// TIA Portal V18 export
// export: Created 2026-01-09T11:31:58.8051596Z, ExportSetting WithDefaults, DisplayName Totally Integrated Automation Portal, DisplayVersion V18 Update 5, DisplayName TIA Portal Openness, DisplayVersion V18 Update 5, DisplayName TIA Portal Teamcenter Gateway, DisplayVersion V18, DisplayName TIA Portal Version Control Interface, DisplayVersion V18, DisplayName SINAMICS Startdrive Advanced, DisplayVersion V18 SP2 Update 1, DisplayName SINAMICS Startdrive G110M, G120, G120C, G120D, G120P, G115D, DisplayVersion V18 SP2 Update 1, DisplayName SINAMICS Startdrive G130, G150, S120, S150, SINAMICS MV, S210, G220, S200, DisplayVersion V18 SP2 Update 1, DisplayName STEP 7 Professional, DisplayVersion V18 Update 5, DisplayName STEP 7 Safety, DisplayVersion V18, DisplayName WinCC Professional, DisplayVersion V18 Update 5
TagTable "GlobalErrorWord"
  GlobalCOMError : Word  (%DB1066.DBW0, CPU S71500-2PN_TP700, 100 ms)
  PNSlaveStation01Error1 : Word  (%DB1066.DBW10, CPU S71500-2PN_TP700, 100 ms)
  PNSlaveStation01Error2 : Word  (%DB1066.DBW12, CPU S71500-2PN_TP700, 100 ms)
  PNSlaveStation01Error3 : Word  (%DB1066.DBW14, CPU S71500-2PN_TP700, 100 ms)
  PNSlaveStation01Error4 : Word  (%DB1066.DBW16, CPU S71500-2PN_TP700, 100 ms)
  PNSlaveStation01Error5 : Word  (%DB1066.DBW18, CPU S71500-2PN_TP700, 100 ms)
  PNSlaveStation01Error6 : Word  (%DB1066.DBW20, CPU S71500-2PN_TP700, 100 ms)
  PNSlaveStation01Error7 : Word  (%DB1066.DBW22, CPU S71500-2PN_TP700, 100 ms)
  PNSlaveStation01Error8 : Word  (%DB1066.DBW24, CPU S71500-2PN_TP700, 100 ms)
  PNSlaveStation01Error9 : Word  (%DB1066.DBW26, CPU S71500-2PN_TP700, 100 ms)
  PNSlaveStation01Error10 : Word  (%DB1066.DBW28, CPU S71500-2PN_TP700, 100 ms)
  SerialCOMM01Error : Word  (%DB1066.DBW30, CPU S71500-2PN_TP700, 100 ms)
  SerialCOMM02Error : Word  (%DB1066.DBW32, CPU S71500-2PN_TP700, 100 ms)
  SerialCOMM03Error : Word  (%DB1066.DBW34, CPU S71500-2PN_TP700, 100 ms)
  SerialCOMM04Error : Word  (%DB1066.DBW36, CPU S71500-2PN_TP700, 100 ms)
  SerialCOMM05Error : Word  (%DB1066.DBW38, CPU S71500-2PN_TP700, 100 ms)
  PNSlaveStation02Error1 : Word  (%DB1066.DBW40, CPU S71500-2PN_TP700, 100 ms)
  PNSlaveStation02Error2 : Word  (%DB1066.DBW42, CPU S71500-2PN_TP700, 100 ms)
  PNSlaveStation02Error3 : Word  (%DB1066.DBW44, CPU S71500-2PN_TP700, 100 ms)
  PNSlaveStation02Error4 : Word  (%DB1066.DBW46, CPU S71500-2PN_TP700, 100 ms)
  PNSlaveStation02Error5 : Word  (%DB1066.DBW48, CPU S71500-2PN_TP700, 100 ms)
  PNSlaveStation02Error6 : Word  (%DB1066.DBW50, CPU S71500-2PN_TP700, 100 ms)
  PNSlaveStation02Error7 : Word  (%DB1066.DBW52, CPU S71500-2PN_TP700, 100 ms)
  PNSlaveStation02Error8 : Word  (%DB1066.DBW54, CPU S71500-2PN_TP700, 100 ms)   // Fault: PLC_OP10_110A1_PNSlaveStationError
  PNSlaveStation02Error9 : Word  (%DB1066.DBW56, CPU S71500-2PN_TP700, 100 ms)
  PNSlaveStation02Error10 : Word  (%DB1066.DBW58, CPU S71500-2PN_TP700, 100 ms)
  PNSlaveStation03Error1 : Word  (%DB1066.DBW60, CPU S71500-2PN_TP700, 100 ms)
  PNSlaveStation03Error2 : Word  (%DB1066.DBW62, CPU S71500-2PN_TP700, 100 ms)
  PNSlaveStation03Error3 : Word  (%DB1066.DBW64, CPU S71500-2PN_TP700, 100 ms)
  PNSlaveStation03Error4 : Word  (%DB1066.DBW66, CPU S71500-2PN_TP700, 100 ms)
  PNSlaveStation03Error5 : Word  (%DB1066.DBW68, CPU S71500-2PN_TP700, 100 ms)
  PNSlaveStation03Error6 : Word  (%DB1066.DBW70, CPU S71500-2PN_TP700, 100 ms)
  PNSlaveStation03Error7 : Word  (%DB1066.DBW72, CPU S71500-2PN_TP700, 100 ms)
  PNSlaveStation03Error8 : Word  (%DB1066.DBW74, CPU S71500-2PN_TP700, 100 ms)
  PNSlaveStation03Error9 : Word  (%DB1066.DBW76, CPU S71500-2PN_TP700, 100 ms)
  PNSlaveStation03Error10 : Word  (%DB1066.DBW78, CPU S71500-2PN_TP700, 100 ms)
  ValveIsland01Error : Word  (%DB1066.DBW80, CPU S71500-2PN_TP700, 100 ms)
  ValveIsland02Error : Word  (%DB1066.DBW82, CPU S71500-2PN_TP700, 100 ms)
  ValveIsland03Error : Word  (%DB1066.DBW84, CPU S71500-2PN_TP700, 100 ms)
  ValveIsland04Error : Word  (%DB1066.DBW86, CPU S71500-2PN_TP700, 100 ms)
  ValveIsland05Error : Word  (%DB1066.DBW88, CPU S71500-2PN_TP700, 100 ms)
  SafetyGlobalError : Word  (%DB1066.DBW90, CPU S71500-2PN_TP700, 100 ms)
  SafetyDoorType01Error : Word  (%DB1066.DBW100, CPU S71500-2PN_TP700, 100 ms)
  SafetyDoorType02Error : Word  (%DB1066.DBW102, CPU S71500-2PN_TP700, 100 ms)
  SafetyDoorType03Error : Word  (%DB1066.DBW104, CPU S71500-2PN_TP700, 100 ms)
  SafetyDoorType04Error : Word  (%DB1066.DBW106, CPU S71500-2PN_TP700, 100 ms)
  SafetyDoorType05Error : Word  (%DB1066.DBW108, CPU S71500-2PN_TP700, 100 ms)
  SafetyDoor01Error : Word  (%DB1066.DBW110, CPU S71500-2PN_TP700, 100 ms)
  SafetyDoor02Error : Word  (%DB1066.DBW112, CPU S71500-2PN_TP700, 100 ms)
  SafetyDoor03Error : Word  (%DB1066.DBW114, CPU S71500-2PN_TP700, 100 ms)
  SafetyDoor04Error : Word  (%DB1066.DBW116, CPU S71500-2PN_TP700, 100 ms)
  SafetyDoor05Error : Word  (%DB1066.DBW118, CPU S71500-2PN_TP700, 100 ms)
  SafetyDoor06Error : Word  (%DB1066.DBW120, CPU S71500-2PN_TP700, 100 ms)
  SafetyDoor07Error : Word  (%DB1066.DBW122, CPU S71500-2PN_TP700, 100 ms)
  SafetyDoor08Error : Word  (%DB1066.DBW124, CPU S71500-2PN_TP700, 100 ms)
  SafetyDoor09Error : Word  (%DB1066.DBW126, CPU S71500-2PN_TP700, 100 ms)
  SafetyDoor10Error : Word  (%DB1066.DBW128, CPU S71500-2PN_TP700, 100 ms)
  LightCurtain01Error : Word  (%DB1066.DBW130, CPU S71500-2PN_TP700, 100 ms)
  LightCurtain02Error : Word  (%DB1066.DBW132, CPU S71500-2PN_TP700, 100 ms)
  LightCurtain03Error : Word  (%DB1066.DBW134, CPU S71500-2PN_TP700, 100 ms)
  LightCurtain04Error : Word  (%DB1066.DBW136, CPU S71500-2PN_TP700, 100 ms)
  LightCurtain05Error : Word  (%DB1066.DBW138, CPU S71500-2PN_TP700, 100 ms)
  Product01Error : Word  (%DB1066.DBW140, CPU S71500-2PN_TP700, 100 ms)
  Product02Error : Word  (%DB1066.DBW142, CPU S71500-2PN_TP700, 100 ms)
  Product03Error : Word  (%DB1066.DBW144, CPU S71500-2PN_TP700, 100 ms)
  Product04Error : Word  (%DB1066.DBW146, CPU S71500-2PN_TP700, 100 ms)
  Product05Error : Word  (%DB1066.DBW148, CPU S71500-2PN_TP700, 100 ms)
  Fixture01Error : Word  (%DB1066.DBW150, CPU S71500-2PN_TP700, 100 ms)
  Fixture02Error : Word  (%DB1066.DBW152, CPU S71500-2PN_TP700, 100 ms)
  Fixture03Error : Word  (%DB1066.DBW154, CPU S71500-2PN_TP700, 100 ms)
  Fixture04Error : Word  (%DB1066.DBW156, CPU S71500-2PN_TP700, 100 ms)
  Fixture05Error : Word  (%DB1066.DBW158, CPU S71500-2PN_TP700, 100 ms)
  Fixture06Error : Word  (%DB1066.DBW160, CPU S71500-2PN_TP700, 100 ms)
  Fixture07Error : Word  (%DB1066.DBW162, CPU S71500-2PN_TP700, 100 ms)
  Fixture08Error : Word  (%DB1066.DBW164, CPU S71500-2PN_TP700, 100 ms)
  Fixture09Error : Word  (%DB1066.DBW166, CPU S71500-2PN_TP700, 100 ms)
  Fixture10Error : Word  (%DB1066.DBW168, CPU S71500-2PN_TP700, 100 ms)
  BreakerTripError01 : Word  (%DB1066.DBW170, CPU S71500-2PN_TP700, 100 ms)
